// TIA Portal V20 export
TYPE "LER_TypeFATMode_Capability_SetValue"
// stored: Access Published
   STRUCT
      SelectCycle_SetValue : Int;
   END_STRUCT;
END_TYPE
